// Brief: Slave Arm test
FUNCTION_BLOCK PUBLIC FB_SlaveCtrlInstruTest EXTENDS FB_SlaveArmCtrlBase
VAR CONSTANT
	m_instruAutoTestTrajNum :INT :=3;
	m_instruVerifyTrajNum :INT :=3;
END_VAR
VAR
	// test mode. 
	//0: stay still; 
	//1: manual joint test ; 
	//2: instrument control verify 
	//3: auto test - finger grip and release
	//4: auto test - finger open and mvoe
	//5: auto test - finger grip and move
	m_instruTestMode :INT := 0;
	m_lastInstruTestMode :INT := 0;
	
	// variables for auto test
	m_autoTestCycles :INT :=0;
	m_autoTestStep :INT :=0;
	m_autoTestTime :LREAL:=0;
	m_instruAutoTestPos:ARRAY [1..m_instruAutoTestTrajNum, 1..3] OF LREAL:=
	[pi/2, 	-135*g_deg2rad,	-45*g_deg2rad,
	 -pi/2,	-15*g_deg2rad, 	60*g_deg2rad,
	 0,		-pi/2, 0];																			
	
	// variable for instument control veify
	m_verifyTestStep :INT :=0;
	m_reachVerifyPos : BOOL := FALSE;
	m_instruVerifyPos:ARRAY [1..m_instruVerifyTrajNum, 1..3] OF LREAL:=
	[pi/2, 	-135*g_deg2rad,	-45*g_deg2rad,
	 -pi/2,	-15*g_deg2rad, 	60*g_deg2rad,
	 0,		-pi/2, 0];		

	// final target DH joint position and grip angle
	m_targetDHJntPos:Vec3d;
	m_targetGripAng:LREAL;
	m_targetGripForceLevel :LREAL :=0;
	
	// interploated command joint position and grip angle 
	m_cmdDHJntPos :Vec6d;
	m_cmdDHJntVel :Vec6d;
	m_cmdGripAng:LREAL;

	// last joint position 
	m_lastCmdJntPos :Vec8d ;
	
	// instrument controller
	m_instruController : FB_BasicInstruControl;
	m_usKnifeController : FB_UltrosonicKnifeControl;
	m_instruCmdJntPos,m_instruCmdJntVel : Vec5d;
	m_instruCmdJntTrq :Vec5d;
	
	// OTG
	m_DHJntOTG:ARRAY[1..3] OF FB_secOrdTrajFilter;
	m_gripAngleOTG : FB_secOrdTrajFilter;
	m_maxJntVel:Vec3d:=[3(2.0)];
	m_maxJntAcc:Vec3d:=[3(4.0)];

END_VAR

METHOD PROTECTED calcCmdJntPos : BOOL
VAR_IN_OUT CONSTANT
	i_endoscopePose : ST_Frame;
	i_masterStatus :ST_MasterStatus;
	i_setupStatus: ST_SetupStatus;
	i_slaveArm :FB_SlaveArm;
END_VAR

VAR 
	i:INT :=0;
	errThres :LREAL;

END_VAR
// determint instrument test mode
m_instruTestMode := determinTestMode();

// determine final target DH joint position
CASE m_instruTestMode OF
	1:
		manualTest(i_slaveArm);
	2:
		instruVerifyTest(i_slaveArm);
	3:
		fingerOpenCloseTest(i_slaveArm);
	4:
		fingerOpenMoveTest(i_slaveArm);
	5:
		fingerGripMoveTest(i_slaveArm);
	ELSE
		m_lastInstruTestMode := m_instruTestMode;
		stayStill(i_slaveArm);
		RETURN;
END_CASE

// run OTG
FOR i:=1 TO 3  DO
	m_DHJntOTG[i].run(m_targetDHJntPos[i],0.0, o_cmdAcc=>,o_cmdVel=>m_cmdDHJntVel[i],o_cmdPos=> m_cmdDHJntPos[i+3]);
END_FOR
m_gripAngleOTG.run(m_targetGripAng,0.0, o_cmdAcc=>,o_cmdVel=>,o_cmdPos=>m_cmdGripAng);

// calculate target motor joint position from DH joint position
i_slaveArm.instrument.instruIK(m_cmdDHJntPos,m_cmdGripAng, o_jntPos=>m_cmdJntPos);

// command velocity
vecSub(m_cmdJntPos, m_lastCmdJntPos, m_cmdJntVel);
vecSelfMultiNum(m_cmdJntVel, g_slaveArmCtrlFreq);
m_lastCmdJntPos:=m_cmdJntPos;

m_lastInstruTestMode := m_instruTestMode;
END_METHOD

// override this function in each exact controller
METHOD PROTECTED calcCmdJntTrq : BOOL
VAR_IN_OUT CONSTANT
	i_endoscopePose : ST_Frame;
	i_masterStatus :ST_MasterStatus;
	i_setupStatus: ST_SetupStatus;
	i_slaveArm :FB_SlaveArm;
END_VAR

VAR 
	nullspaceMat :Mat7d;
	ctrlTrq : Vec7d;
	i : int ;
END_VAR
// set joint torque to zero in default
m_cmdJntTrq := g_zeroVec8d;

// instrument joint control
FOR i:=1 TO 5 DO 
	m_instruCmdJntPos[i]:=m_cmdJntPos[i+3];
	m_instruCmdJntVel[i]:=m_cmdJntVel[i+3];
END_FOR

IF i_slaveArm.instrument.instruType = InstruType_UltrasoundKnifeS OR i_slaveArm.instrument.instruType = InstruType_UltrasoundKnifeU THEN
	m_usKnifeController.run(m_instruCmdJntPos,m_instruCmdJntVel, m_targetGripForceLevel, i_slaveArm, o_cmdJntTrq=>m_instruCmdJntTrq);
ELSE
	m_instruController.run(m_instruCmdJntPos,m_instruCmdJntVel, m_cmdDHJntPos[6], m_cmdDHJntVel[6], m_targetGripForceLevel, i_slaveArm, o_cmdJntTrq=>m_instruCmdJntTrq);
END_IF

FOR i:=1 TO 5 DO
	m_cmdJntTrq[i+3]:=m_instruCmdJntTrq[i];
END_FOR
END_METHOD

METHOD determinTestMode : INT
VAR_INPUT
END_VAR
determinTestMode :=0;
IF GVL_InstruTestUIVars.g_instruManulTestFlag THEN
	determinTestMode := 1;
END_IF;

IF GVL_InstruTestUIVars.g_instruPosVerifyFlag THEN
	determinTestMode := 2;
ELSE
	m_verifyTestStep :=0;
END_IF

IF GVL_InstruTestUIVars.g_instruAutoTestFlag THEN
	determinTestMode := GVL_InstruTestUIVars.g_instruAutoTestMode +3; 
ELSE
	m_autoTestCycles := 0;
	m_autoTestStep :=0;
END_IF
END_METHOD

METHOD fingerGripMoveTest : BOOL
VAR_IN_OUT CONSTANT
	i_slaveArm :FB_SlaveArm;
END_VAR
VAR
	i:INT;
END_VAR
m_targetGripForceLevel :=100;
m_autoTestStep := LIMIT(0,m_autoTestStep, m_instruAutoTestTrajNum-1);
FOR i:=1 TO 3 DO
	 m_targetDHJntPos[i] := m_instruAutoTestPos[m_autoTestStep+1, i];
END_FOR
	 
IF ABS(m_cmdDHJntPos[4]-m_targetDHJntPos[1])< g_jntCtrlAngTolLow AND ABS(m_cmdDHJntPos[5]-m_targetDHJntPos[2])< g_jntCtrlAngTolLow 
		AND ABS(m_cmdDHJntPos[6]-m_targetDHJntPos[3])< g_jntCtrlAngTolLow  THEN
	m_autoTestStep :=m_autoTestStep + 1;
END_IF
 
IF m_autoTestStep >= m_instruAutoTestTrajNum THEN
	m_autoTestCycles := m_autoTestCycles + 1;
	m_autoTestStep := 0;
END_IF
END_METHOD

METHOD fingerOpenCloseTest : BOOL
VAR_IN_OUT CONSTANT
	i_slaveArm :FB_SlaveArm;
END_VAR
m_targetGripForceLevel :=0;
m_autoTestStep := LIMIT(0,m_autoTestStep, 1);
IF m_autoTestStep =0 THEN
	m_targetGripAng := i_slaveArm.instrument.kinematicParameters.m_maxGripAngle;
ELSE
	m_targetGripAng := 0;
END_IF
m_targetDHJntPos[1] := 0;
m_targetDHJntPos[2] := -pi/2;
m_targetDHJntPos[3] := 0;

IF ABS(m_cmdGripAng- m_targetGripAng)< g_jntCtrlAngTolLow THEN
	 m_autoTestStep :=m_autoTestStep + 1;
END_IF

IF m_autoTestStep > 1 THEN
	m_autoTestCycles := m_autoTestCycles + 1;
	m_autoTestStep := 0;
END_IF
END_METHOD

METHOD fingerOpenMoveTest : BOOL
VAR_IN_OUT CONSTANT
	i_slaveArm :FB_SlaveArm;
END_VAR
VAR
	i:INT;
END_VAR
m_targetGripForceLevel :=0;
m_autoTestStep := LIMIT(0,m_autoTestStep, m_instruAutoTestTrajNum-1);
FOR i:=1 TO 3 DO
	 m_targetDHJntPos[i] := m_instruAutoTestPos[m_autoTestStep+1, i];
END_FOR
	 
IF ABS(m_cmdDHJntPos[4]-m_targetDHJntPos[1])< g_jntCtrlAngTolLow AND ABS(m_cmdDHJntPos[5]-m_targetDHJntPos[2])< g_jntCtrlAngTolLow 
		AND ABS(m_cmdDHJntPos[6]-m_targetDHJntPos[3])< g_jntCtrlAngTolLow  THEN
	m_autoTestStep :=m_autoTestStep + 1;
END_IF
 
IF m_autoTestStep >= m_instruAutoTestTrajNum THEN
	m_autoTestCycles := m_autoTestCycles + 1;
	m_autoTestStep := 0;
END_IF
END_METHOD

METHOD PUBLIC init : BOOL
VAR_IN_OUT CONSTANT
	i_slaveArm	:FB_SlaveArm;
END_VAR
VAR_IN_OUT 
	r_slaveArmCtrlCmd :ST_SlaveArmCtrlCmds;
END_VAR

VAR
	i:int;
END_VAR
SUPER^.Init(i_slaveArm,r_slaveArmCtrlCmd);
m_lastCmdJntPos:=m_cmdJntPos;
m_jntOPMode[1] := DriverOPMode_PosTrq;
m_jntOPMode[2] := DriverOPMode_PosTrq;
m_jntOPMode[3] := DriverOPMode_PosTrq;
m_jntOPMode[4] := DriverOPMode_Trq;
m_jntOPMode[5] := DriverOPMode_Trq;
m_jntOPMode[6] := DriverOPMode_Trq;
m_jntOPMode[7] := DriverOPMode_Trq;
m_jntOPMode[8] := DriverOPMode_Trq;

m_cmdDHJntPos :=i_slaveArm.curDHJntPos;
m_cmdDHJntVel :=g_zeroVec6d;
m_targetGripAng := i_slaveArm.curGripAngle;
m_targetDHJntPos[1] := i_slaveArm.curDHJntPos[4];
m_targetDHJntPos[2] := i_slaveArm.curDHJntPos[5];
m_targetDHJntPos[3] := i_slaveArm.curDHJntPos[6];

// init instrument controller
m_instruController.init(i_slaveArm);
m_usKnifeController.init(i_slaveArm);

FOR i:=1 TO 3  DO
	m_DHJntOTG[i].init(m_cmdDHJntPos[i+3], 0, m_maxJntVel[i], m_maxJntAcc[i], g_slaveArmCtrlCycleTime);
END_FOR

m_gripAngleOTG.init(m_targetGripAng, 0, 2*m_maxJntVel[3], 2*m_maxJntAcc[3], g_slaveArmCtrlCycleTime);
// update commands to arm
copyCmds(r_slaveArmCtrlCmd);
END_METHOD

METHOD instruVerifyTest : BOOL
VAR_IN_OUT CONSTANT
	i_slaveArm :FB_SlaveArm;
END_VAR
VAR
	i:INT;
END_VAR
m_targetGripForceLevel :=0;
m_autoTestStep := LIMIT(0,m_autoTestStep, m_instruVerifyTrajNum-1);
IF m_verifyTestStep = 0 THEN
	m_targetGripAng := i_slaveArm.instrument.kinematicParameters.m_maxGripAngle;
ELSE
	m_targetGripAng := 0;
END_IF

FOR i:=1 TO 3 DO
	 m_targetDHJntPos[1] := m_instruVerifyPos[m_verifyTestStep+1, i];
END_FOR
	 
m_reachVerifyPos := ABS(m_cmdDHJntPos[4]-m_targetDHJntPos[1])< g_jntCtrlAngTolLow AND ABS(m_cmdDHJntPos[5]-m_targetDHJntPos[2])< g_jntCtrlAngTolLow 
		AND ABS(m_cmdDHJntPos[6]-m_targetDHJntPos[3])< g_jntCtrlAngTolLow ; 

IF  GVL_InstruTestUIVars.g_instruPosVerifyNextStepFlag THEN
	m_verifyTestStep :=m_verifyTestStep + 1;
ELSIF  GVL_InstruTestUIVars.g_instruPosVerifyLastStepFlag THEN
	m_verifyTestStep :=m_verifyTestStep - 1;
END_IF
END_METHOD

METHOD manualTest : BOOL
VAR_IN_OUT CONSTANT
	i_slaveArm :FB_SlaveArm;
END_VAR
IF GVL_InstruTestUIVars.g_moveToSetPosFlag THEN
	m_targetDHJntPos[1] := GVL_InstruTestUIVars.g_targetRollAng*g_deg2rad;
	m_targetDHJntPos[2] := GVL_InstruTestUIVars.g_targetPitchAng*g_deg2rad;
	m_targetDHJntPos[3] := GVL_InstruTestUIVars.g_targetYawAng*g_deg2rad;
	m_targetGripAng := GVL_InstruTestUIVars.g_targetGripAng*g_deg2rad;
	m_targetGripForceLevel := LIMIT(0, GVL_InstruTestUIVars.g_targetGripForceLevel, 100);
ELSIF GVL_InstruTestUIVars.g_gripperOpenFlag THEN
	m_targetGripAng := i_slaveArm.instrument.kinematicParameters.m_maxGripAngle;
	m_targetGripForceLevel :=0;
ELSIF GVL_InstruTestUIVars.g_gripperCloseFlag THEN
	m_targetGripAng := 0;
	m_targetGripForceLevel :=0;
ELSIF GVL_InstruTestUIVars.g_maxGripForceFlag THEN
	m_targetGripAng := 0;
	m_targetGripForceLevel :=100;
END_IF
END_METHOD

METHOD stayStill : BOOL
VAR_IN_OUT CONSTANT
	i_slaveArm :FB_SlaveArm;
END_VAR
VAR
	i:int;
END_VAR
IF m_lastInstruTestMode>=1 AND m_lastInstruTestMode <5 THEN
	m_cmdJntPos := i_slaveArm.curJntPos;
END_IF
m_cmdJntVel := g_zeroVec8d;
m_lastCmdJntPos := m_cmdJntPos;
m_cmdDHJntPos :=i_slaveArm.curDHJntPos;
m_cmdDHJntVel :=g_zeroVec6d;
m_targetGripAng := i_slaveArm.curGripAngle;
m_targetGripForceLevel := 0;

FOR i:=1 TO 3  DO
	m_DHJntOTG[i].init(m_cmdDHJntPos[i+3], 0, m_maxJntVel[i], m_maxJntAcc[i], g_slaveArmCtrlCycleTime);
END_FOR

m_gripAngleOTG.init(m_targetGripAng, 0, 2*m_maxJntVel[3], 2*m_maxJntAcc[3], g_slaveArmCtrlCycleTime);
END_METHOD

END_FUNCTION_BLOCK

(* stored: Version 1.1.0.1, ProductVersion 3.1.4024.11
   POU FB_SlaveCtrlInstruTest: Id {d70115e7-7668-49fd-9f57-bdf3458ba446}, SpecialFunc None
   Method calcCmdJntPos: Id {fabdb455-5225-4307-a367-b36816d27b6f}
   Method calcCmdJntTrq: Id {89cc8590-b0ea-4a29-944b-9b994680a8df}
   Method determinTestMode: Id {873d96b2-7877-4cfa-9ab1-26e8410379b0}
   Method fingerGripMoveTest: Id {b23b170a-3eed-478e-a97c-17d1ca24b714}
   Method fingerOpenCloseTest: Id {7cc8daed-3bf9-42ca-9d17-f827b074e621}
   Method fingerOpenMoveTest: Id {9c6e0ab8-ec0f-4e57-8c89-55d8aad6317c}
   Method init: Id {1224d61d-417a-4654-acf9-99ef0220f449}
   Method instruVerifyTest: Id {32fd7dea-b530-44b3-81c2-23f19fa7b97f}
   Method manualTest: Id {35aef409-4f2b-4e32-b983-7a5a4b214e71}
   Method stayStill: Id {d0e64cf1-810c-48a9-bb08-c3a957da86ae} *)
